Staubli VAL3: page_changeTrsf.pgx

public program page_changeTrsf(trsf& x_tTrsf[], bool x_bUseFrame, bool x_bUseReset, string x_sTitle, string x_sComment)
  local string l_sEvent
  local num l_nFrame
  local num l_nView
  local bool l_bRefresh
  local bool l_bTest
  local num l_nKey
  local num i
  local string l_sMessage
  local trsf l_tTrsf
  local string l_sItem
  local string l_sEmpty
begin
  logMsg("[KERNEL] INTERFACE:PAGE changeTrsf "+x_sTitle)
  l_bRefresh=false
  l_nFrame=0
  l_nView=0
  call use:setSizeList(19,0,19,8)
  call use:setView(false)
  l_tTrsf=x_tTrsf
  //
  do
    cls()
    call use:type(0,12,x_sComment)
    call use:typeMenu(8,"OK")
    if x_bUseReset
      call language:message(l_sMessage,184)
      call use:strfill(l_sMessage,5,l_sMessage)
      call use:type(21,13,l_sMessage)
    endIf
    call use:listcreate(x_sTitle)
    l_sItem="coord  X > "+toString(".3",l_tTrsf.x)
    call use:listadd(l_sItem)
    l_sItem="coord  Y > "+toString(".3",l_tTrsf.y)
    call use:listadd(l_sItem)
    l_sItem="coord  Z > "+toString(".3",l_tTrsf.z)
    call use:listadd(l_sItem)
    l_sItem="coord RX > "+toString(".3",l_tTrsf.rx)
    call use:listadd(l_sItem)
    l_sItem="coord RY > "+toString(".3",l_tTrsf.ry)
    call use:listadd(l_sItem)
    l_sItem="coord RZ > "+toString(".3",l_tTrsf.rz)
    call use:listadd(l_sItem)
    use:nView=l_nFrame
    call use:listupdate(l_nFrame-l_nView)
    do
      l_nView=use:nView
      l_nKey=get()
      call use:listevent(l_nKey,l_nFrame,l_sEvent)
      switch l_nKey
        case 270
          //
          // clean the line
          call use:listcursor(use:nView,false)
          switch l_nFrame
            case 0
              //  x-value
              call use:changeValue(l_tTrsf.x,0,0,10+40-use:nBottomX,use:nView+1,l_sEmpty)
            break
            case 1
              //  y-value
              call use:changeValue(l_tTrsf.y,0,0,10+40-use:nBottomX,use:nView+1,l_sEmpty)
            break
            case 2
              //  z-value
              call use:changeValue(l_tTrsf.z,0,0,10+40-use:nBottomX,use:nView+1,l_sEmpty)
            break
            case 3
              //  rx-value
              call use:changeValue(l_tTrsf.rx,0,0,10+40-use:nBottomX,use:nView+1,l_sEmpty)
            break
            case 4
              //  ry-value
              call use:changeValue(l_tTrsf.ry,0,0,10+40-use:nBottomX,use:nView+1,l_sEmpty)
            break
            case 5
              //  rz-value
              call use:changeValue(l_tTrsf.rz,0,0,10+40-use:nBottomX,use:nView+1,l_sEmpty)
            break
          endSwitch
          l_bRefresh=true
        break
        case 278
          // VALIDATE
          x_tTrsf=l_tTrsf
        break
        case 275
          // RESET
          if x_bUseReset
            l_tTrsf={0,0,0,0,0,0}
            l_bRefresh=true
          endIf
        break
      endSwitch
    until l_bRefresh==true or l_nKey==255 or l_nKey==278
    l_bRefresh=false
  until l_nKey==255 or l_nKey==278
  // release the resource
  call use:nullKey(l_nKey)
  if !cycleStatus:bCycle and !cycleStatus:bSimulation
    resetMotion()
  endIf
end
